# EPICS substitutions: iocBoot/ioc13ida/13ID_BPM_Foil.substitutions
file "$(CARS)/db/13ID_BPM_Foil.template"
{
pattern
{P,      R,      MOTOR, F1,   F2, F3, F4, F5, F6}
# Old foils (pre-2015)
#{13IDA:, CD_BPM, m34,   Open, Ti, Cr, Ni, Cu, Empty}
#{13IDA:, E_BPM,  m33,   Open, Ti, Cr, Ni, Cu, Empty}
# New foils (as of 2015 run 1)
{13IDA:, CD_BPM, m34,   Open, Ti, Ag, Ni, Cu, Au}
{13IDA:, E_BPM,  m33,   Open, Ti, Cr, Ni, Al, Au}
}
